FUNCTION_BLOCK MapAndPath (* Tamplate for a simple Basic Function Block Type *)
  (* Standard: 61499-2 *)
  (* Version 0.0, 2018-06-04, 4DIAC-IDE, 4DIAC-Consortium *)
  (* Version 1.0, 2016-05-26, AZ, fortiss GmbH *)
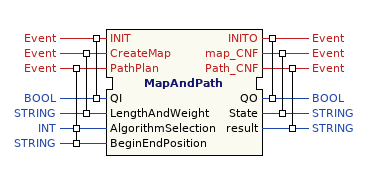
  EVENT_INPUT
    INIT WITH QI; (* Initialization Request *)
    CreateMap WITH LengthAndWeight; (* Normal Execution Request *)
    PathPlan WITH AlgorithmSelection, BeginEndPosition;
  END_EVENT
  EVENT_OUTPUT
    INITO WITH QO; (* Initialization Confirm *)
    map_CNF WITH State; (* Execution Confirmation *)
    Path_CNF WITH result;
  END_EVENT
  VAR_INPUT
    QI : BOOL; (* Input event qualifier *)
    LengthAndWeight : STRING; (* msg frame：Length_Weight *)
    AlgorithmSelection : INT; (* 1-Dijkstra, 2-others reservation *)
    BeginEndPosition : STRING; (* like 1_10 *)
  END_VAR
  VAR_OUTPUT
    QO : BOOL; (* Output event qualifier *)
    State : STRING; (* Creat map success or failed *)
    result : STRING; (* like 1-->3-.... *)
  END_VAR
  VAR
    maxNum : INT; (* Internal Variable *)
  END_VAR
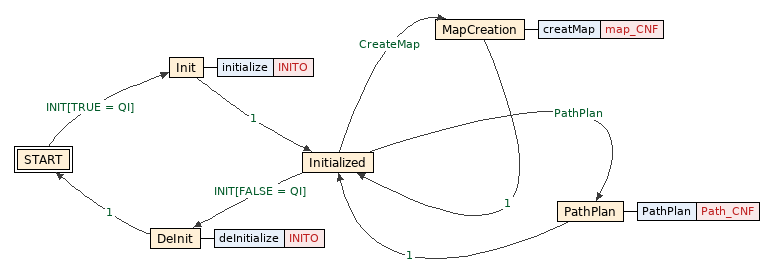
  EC_STATES
    START; (* Initial State *)
    Init : initialize -> INITO; (* Initialization *)
    MapCreation : creatMap -> map_CNF; (* Normal execution *)
    Initialized;
    DeInit : deInitialize -> INITO;
    PathPlan : PathPlan -> Path_CNF;
  END_STATES
  EC_TRANSITIONS
    START TO Init := INIT[TRUE = QI];
    Init TO Initialized := 1;
    Initialized TO MapCreation := CreateMap;
    MapCreation TO Initialized := 1;
    DeInit TO START := 1;
    Initialized TO DeInit := INIT[FALSE = QI];
    Initialized TO PathPlan := PathPlan;
    PathPlan TO Initialized := 1;
  END_TRANSITIONS
  ALGORITHM initialize IN ST: (* Initialization algorithm *)
QO := QI;
  END_ALGORITHM
  ALGORITHM deInitialize IN ST: (* Normally executed algorithm *)
QO := FALSE;
  END_ALGORITHM
  ALGORITHM creatMap IN ST: (* new algorithm *)
LengthAndWeight:="hfrhkd";
State:="OK";
  END_ALGORITHM
  ALGORITHM PathPlan IN ST: (* new algorithm *)
AlgorithmSelection:=1;
BeginEndPosition:="1_10";
result:="1-2-3";
maxNum:=100;
  END_ALGORITHM
END_FUNCTION_BLOCK
